FUNCTION_BLOCK DegreesToRelativeMovment
VAR_INPUT
	MaxRelativePoint : LREAL;
	MaxSteeringAngle : INT;
	Deg : LREAL;
END_VAR
VAR_OUTPUT
	RelativeMovement : LREAL;
END_VAR
VAR
END_VAR

//IF (Deg > 0 OR Deg < 0) THEN
	RelativeMovement := (MaxRelativePoint/MaxSteeringAngle)*Deg;
//ELSIF (Deg = 0) THEN
	//RelativeMovement := MaxRelativePoint/2;		
//END_IF

END_FUNCTION_BLOCK

(* stored: Version 1.1.0.1, ProductVersion 3.1.4024.3
   POU DegreesToRelativeMovment: Id {cd224430-36b7-483d-b332-e0d072bad6ee}, SpecialFunc None *)
